TYPE A21ToolStorage :
STRUCT
	pos1ChipboardEOAT AT %I* : BOOL;
	pos1WoodBunkEOAT AT %I* : BOOL;
	
	pos2ChipboardEOAT AT %I* : BOOL;
	pos2WoodBunkEOAT AT %I* : BOOL;
END_STRUCT
END_TYPE

(* stored: Version 1.1.0.1, ProductVersion 3.1.4024.11
   DUT A21ToolStorage: Id {f35f457f-7778-4b2a-a585-ad4ff14a5f49} *)
